(* CODESYS project MethodsExport.export

Project tree, tasks and I/O mapping:
  program Main [ST]
  function block Motor [ST]: Start, Stop
*)

// Main
PROGRAM Main
VAR_INPUT
	MotorA : Motor;
	methodHasCompleted : BOOL;
END_VAR


// Call a method and get the return value

methodHasCompleted := MotorA.Start();

END_PROGRAM

// Motor
FUNCTION_BLOCK Motor
VAR
	MotorRunOutput : BOOL;
END_VAR

METHOD Start : BOOL

// Check motor is ok to start then...

MotorRunOutput := TRUE;

// Return a value
Start := TRUE;
END_METHOD

METHOD Stop : BOOL

// Check motor is ok to stop then...

MotorRunOutput := FALSE;
END_METHOD

END_FUNCTION_BLOCK
